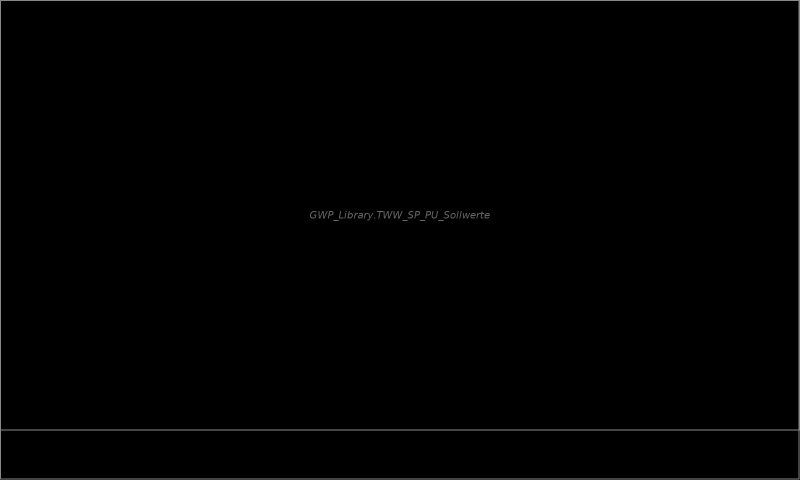
VISUALIZATION TWW_SP_PU_Sollwerte  // 800x480
    Frame (0,0 800x430)
        shows GWP_Library.TWW_SP_PU_Sollwerte(FB_TWW_SP := Main.TWW_SP_0, FB_Init_1 := Main.Init_0)
END_VISUALIZATION

(* stored: Version 1.1.0.1, ProductVersion 3.1.4022.6
   Visu TWW_SP_PU_Sollwerte: Id {95999637-2512-4dda-bab7-2f27e1654b0e} *)
